(* PLC project LiquidLevelControler.project, CODESYS CODESYS V3.5 SP10 *)
(* stored: creationDateTime 2018-02-17T15:27:48.2946018, modificationDateTime 2018-02-17T15:27:33.3769123 *)

PROGRAM Main
  VAR_INPUT
    START : BOOL;
    STOP : BOOL;
    LSL_1 : BOOL;
    LSH_1 : BOOL;
  END_VAR
  VAR_OUTPUT
    AUTO : BOOL;
    PUMP : BOOL;
  END_VAR

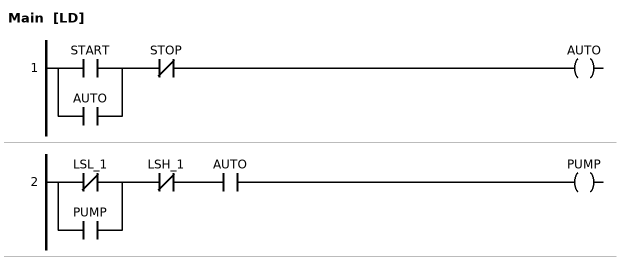
(* LD diagram, written out as Structured Text *)

AUTO := (START OR AUTO) AND NOT STOP;

PUMP := (NOT LSL_1 OR PUMP) AND NOT LSH_1 AND AUTO;
END_PROGRAM

CONFIGURATION Application
  RESOURCE Application ON PLC
    TASK Task(INTERVAL := T#20ms, PRIORITY := 1);
    PROGRAM Main WITH Task : Main;
  END_RESOURCE
END_CONFIGURATION
